Fanuc KAREL source: kt00811.KL

-- PROVISIONAL review KL for V770-1; original PC SHA256 c36d83ff4f5396a0d8d7b291d5b2127426a8e423466b490da42636feaf67e9f7
-- Incomplete behavior may be omitted. Consult companion uncertainty JSON. Do not deploy.
PROGRAM KT00811
%NOLOCKGROUP
VAR
  R1 : REAL
  R2 : REAL
  OUT : REAL
BEGIN
  -- UNRESOLVED_PC offsets 5-16; opcodes 2E,23
  -- UNRESOLVED_PC offsets 21-32; opcodes 2E,23
  -- UNRESOLVED_PC offsets 37-48; opcodes 2E,23
  -- UNRESOLVED_PC offsets 53-64; opcodes 2E,23
  -- UNRESOLVED_PC offsets 69-84; opcodes 27,22,76,23
  -- UNRESOLVED_PC offsets 89-93; opcodes 7F
END KT00811
